FUNCTION_BLOCK FB_TIIAlarm
VAR_INPUT
	vIO							: ST_TCMultiLevel_VIO;
	stTCColVIO					: ST_TCColumn_VIO;
	NoOfTIIAlm					: INT	:= NO_OF_TII_SENSOR;
	iLevel						: INT	:= 1;
END_VAR

VAR_OUTPUT
	isTIIError					: BOOL;
	TIIAlarmLED					: BOOL;
	TIIAlarmEPT					: BOOL;
	iUnBlock					: DINT;
	isAboveCellLeakage			: BOOL;
END_VAR

VAR
	DIFU						: R_TRIG;
	tim							: TON;
	delay						: FB_Delay;
	tPOn						: BOOL;	//testerPowerOutoutOn after Delay
	dPOn						: BOOL; //dpsPwrbit after Delay
	bitNo						: INT;
	almRset						: BOOL;
	
	ArrAlmBitBefDelay			: ARRAY[1..NO_OF_TII_SENSOR] OF BOOL;
	ArrAlmBitAftDelay			: ARRAY[1..NO_OF_TII_SENSOR] OF BOOL;
	ArrAlarmKeepBit				: ARRAY[1..NO_OF_TII_SENSOR] OF BOOL;
	ArrDelayAlarm				: ARRAY[1..NO_OF_TII_SENSOR] OF FB_AlarmDelay;
	Arr_ms						: ARRAY[1..NO_OF_TII_SENSOR] OF INT;
	bTIIByPassArray				: ARRAY[1..NO_OF_TII_SENSOR] OF BOOL;
	i							: INT;
	bTest						: BOOL;
	delayExtTimeOut				: FB_Delay;
	delayRetTimeOut				: FB_Delay;
	delayDrawerUpTimeOut		: FB_Delay;
	delayDrawerDownTimeOut		: FB_Delay;
	//iUnBlock:INT;
	alarmReset					: BOOL;  //1: reset timer when alarm reset, 0: do not reset timer
END_VAR

VAR_IN_OUT
	
	//bLibError : BOOL;
	//stAlmSubMod:ST_AlarmSubmodules;
	//stAlmMod:ST_AlarmModules;
END_VAR

//<HMI_TII_Test>

IF bHMITIIBypass THEN
	bTIIByPassArray							:= stHMITIIByPassArray[iLevel].bHMITIIByPassArray;
	//FOR i:=1 TO NoOfTIIAlm DO
	//	bTIIByPassArray[i]:= NOT stHMITIIByPassArray[iLevel].bHMITIIByPassArray[i];
	//END_FOR
ELSE
	FOR i := 1 TO NoOfTIIAlm DO
		//bTIIByPassArray[i]:=bEnableTIIAlarm;
		 bTIIByPassArray[i]					:= TC_ModuleState[iLevel].TCSite[1].TIERII = E_State.eEnabled;
	END_FOR
END_IF
//</HMI_TII_Test>
//IF bTest THEN
AlarmUpdate(bENs:= bTIIByPassArray);
//END_IF

METHOD AlarmUpdate : BOOL
VAR_INPUT
	bENs 					: ARRAY [1..NO_OF_TII_SENSOR] OF BOOL;
END_VAR

VAR_OUTPUT
END_VAR

VAR_IN_OUT
	//ArrAlarmKeepBit:ST_AlarmTags;
END_VAR

VAR
	_bError					: BOOL;
	bTstOnCmd 				: BOOL;
	bChkTstOn 				: BOOL;
	bAPOnCmd				: BOOL;
	bChkAPOn 				: BOOL;
	drawerExtendOutput		: BOOL; // Condition
	drawerRetractOutput		: BOOL; // Condition
	drawerUpOutput			: BOOL;
	drawerDownOutput		: BOOL;
	
	i						: INT;
	j						: INT;
	iSysAlarmID 			: INT;
	e						: E_TIIAlarm;
END_VAR
IF iLevel = 0 THEN
	RETURN;
END_IF

//FB_M_nCyclic_tSensorTimeOut
DIFU(
	CLK 																:= vIO.ipTesterPowerOn);
	                                                					
tim(                                                					
	IN 																	:= TRUE,
	PT																	:= INT_TO_TIME(1000));
	                                                					
tPOn 																	:=	VIO.bTstDelInt; //Delay and TesterPwrOnOutput
                                                    					
delay(                                              					
	msec 																:= 100,
	in 																	:= tPOn, 
	out 																:= dPOn);
	                                                					
delayExtTimeOut(                                    	
	msec																:= TIME_TO_INT(tDwrCylExtRetTimeOut),
	in																	:= vIO.opCellDrawerCylExtend,
	out																	:= drawerExtendOutput);
	                                                					
delayRetTimeOut(                                    					
	msec																:= TIME_TO_INT(tDwrCylExtRetTimeOut),
	in																	:= vIO.opCellDrawerCylRetract,
	out																	:= drawerRetractOutput);
	

delayDrawerUpTimeOut(
	msec																:= TIME_TO_INT(tDwrCylUpDownTimeOut),
	in																	:= vIO.opCellDrawerCylUp,
	out																	:= drawerUpOutput);

delayDrawerDownTimeOut(
	msec																:= TIME_TO_INT(tDwrCylUpDownTimeOut),
	in																	:= vIO.opCellDrawerCylDown,
	out																	:= drawerDownOutput);
	

//lRt:= FALSE; //:=AP_Deactuated(if AP Down Can Retract)
//lEt:= FALSE;
bTstOnCmd																:= vIO.bDPSPowerOnOff;
bChkTstOn																:= vIO.bChkTesterOn;
bAPOnCmd																:= vIO.bAP240ACPowerOnOff;
bChkAPOn																:= vIO.bChkAP240On;


//Auto reset Door lock alarm
IF ALMTC.Level[iLevel].AlarmID[E_TIIAlarm.ipTCCellDoorClosed] AND vIO.ipTCCellDoorClosed THEN
	ALMTC.Level[iLevel].AlarmID[E_TIIAlarm.ipTCCellDoorClosed]			:= FALSE;
END_IF

IF ALMTC.Level[iLevel].AlarmID[E_AlarmID.DoorCloseSignalNotDetected] AND vIO.ipTCCellDoorOpenCloseStatus THEN
	ALMTC.Level[iLevel].AlarmID[E_AlarmID.DoorCloseSignalNotDetected]			:= FALSE;
END_IF

//Auto reset Door lock alarm (Debugcart only)
IF bDebugCart THEN
	//auto clear alarm if door is closed 
	IF ALMTC.Level[iLevel].AlarmID[E_AlarmID.TBotSideDoorCloseSignalNotDetected] THEN
		IF VIO.ipTCCellTbotSideDoorOpenCloseStatus01 AND VIO.ipTCCellTbotSideDoorOpenCloseStatus02 THEN
			ALMTC.Level[iLevel].AlarmID[E_AlarmID.TBotSideDoorCloseSignalNotDetected]		:= FALSE;
		END_IF
	END_IF
	
	//auto clear alarm if door is locked
	IF ALMTC.Level[iLevel].AlarmID[E_TIIAlarm.FrontDoorLockSignalNotDetected] THEN
		IF VIO.ipTCCellTbotSideDoorLocked01 AND VIO.ipTCCellTbotSideDoorLocked02 THEN
			ALMTC.Level[iLevel].AlarmID[E_TIIAlarm.FrontDoorLockSignalNotDetected]		:= FALSE;
		END_IF
	END_IF
END_IF


FOR i := 1 TO NoOfTIIAlm DO	
	CASE i OF
		(*E_TIIAlarm.ipAPPresentSensor: 
			e															:= E_TIIAlarm.ipAPPresentSensor; 
			ArrAlmBitBefDelay[E_TIIAlarm.ipAPPresentSensor]				:= (NOT	vIO.ipAPPresentSensor) AND bENs[1];  		
			Arr_ms[e] 													:= 500;  (*TIIAlmText[e]:='AP_PresentSensor'*); //****stTCVIO.iAlarmCode=  E_Alarm.ipAP_PresentSensor 	 ;*)
			
        E_TIIAlarm.ipAPPowerOn: 
			e															:= E_TIIAlarm.ipAPPowerOn; 
			ArrAlmBitBefDelay[E_TIIAlarm.ipAPPowerOn]					:= (NOT vIO.ipAPPowerOn) AND VIO.ipAPPresentSensor AND GVL_DUT_TC_AP240ACPower.Failed AND bENs[2];
			Arr_ms[e] 													:= 500;  (*TIIAlmText[e]:='AP_PowerOn'*); 
			
	    E_TIIAlarm.ipAPReady: 
			e															:= E_TIIAlarm.ipAPReady; 
			ArrAlmBitBefDelay[E_TIIAlarm.ipAPReady]						:= (NOT vIO.ipAPReady) AND vIO.ipAPPresentSensor AND bENs[3]; 	
			Arr_ms[e] 													:= 500;  (*TIIAlmText[e]:='AP_Ready' 		    	*);      
			
	    (*E_TIIAlarm.ipAPDeactuatedPLC: 
			e															:= E_TIIAlarm.ipAPDeactuatedPLC; 
			ArrAlmBitBefDelay[E_TIIAlarm.ipAPDeactuatedPLC]				:= (NOT vIO.ipHandlerSafeToEnterPLC) AND vIO.ipAPPresentSensor AND bENs[4]; 			
			Arr_ms[e] 													:= 500;  (*TIIAlmText[e]:='AP_DeactuatedPLC'*); *)
  
	    (*E_TIIAlarm.ipAPDeactuatedHwr: 
			e															:= E_TIIAlarm.ipAPDeactuatedHwr; 
			ArrAlmBitBefDelay[E_TIIAlarm.ipAPDeactuatedHwr]				:= (NOT	vIO.ipHandlerSafeToEnterHwr) AND vIO.ipAPPresentSensor AND bENs[5]; 			
			Arr_ms[e] 													:= 500;  (*TIIAlmText[e]:='AP_DeactuatedHwr'*); *)
			
	    E_TIIAlarm.ipCellFluidLeakage1: 
			e															:= E_TIIAlarm.ipCellFluidLeakage1; 
			ArrAlmBitBefDelay[E_TIIAlarm.ipCellFluidLeakage1]			:= vIO.ipCellFluidLeakage1 (*AND bENs[6]*); 			
			Arr_ms[e] 													:= 500;  (*TIIAlmText[e]:='CellFluidLeakage1' 	*);   
			
	    E_TIIAlarm.ipCellFluidLeakage2: 
			e															:= E_TIIAlarm.ipCellFluidLeakage2; 
			ArrAlmBitBefDelay[E_TIIAlarm.ipCellFluidLeakage2]			:= vIO.ipCellFluidLeakage2 (*AND bENs[7]*) ; 			
			Arr_ms[e] 													:= 500;  (*TIIAlmText[e]:='CellFluidLeakage2'*);   
			
	    E_TIIAlarm.ipCellGroundFault: 
			e															:= E_TIIAlarm.ipCellGroundFault; 
			ArrAlmBitBefDelay[E_TIIAlarm.ipCellGroundFault]				:= vIO.ipCellGroundFault AND bENs[8]; 			
			Arr_ms[e] 													:= 500;  (*TIIAlmText[e]:='CellGroundFault'*);
			
        (*E_TIIAlarm.ipTesterPresent: 
			e															:= E_TIIAlarm.ipTesterPresent; 
			ArrAlmBitBefDelay[E_TIIAlarm.ipTesterPresent]				:= (NOT	vIO.ipTesterPresent) AND bENs[9]; 			
			Arr_ms[e] 													:= 500;  (*TIIAlmText[e]:='TesterPresent'*);*)
			
        E_TIIAlarm.ipTesterPowerOn: 
			e															:= E_TIIAlarm.ipTesterPowerOn; 
			ArrAlmBitBefDelay[E_TIIAlarm.ipTesterPowerOn]				:= (NOT	vIO.ipTesterPowerOn) AND vIO.ipTesterPresent AND bChkTstOn AND bENs[10]; 			
			Arr_ms[e] 													:= 500;  (*TIIAlmText[e]:='TesterPowerOn'*);
    
        (*E_TIIAlarm.ipTesterReady: 
			e															:= E_TIIAlarm.ipTesterReady; 
			ArrAlmBitBefDelay[E_TIIAlarm.ipTesterReady]					:= (NOT	vIO.ipTesterReady) AND vIO.ipTesterPresent AND bENs[11]; 	
			Arr_ms[e] 													:= 500;  (*TIIAlmText[e]:='TesterReady'*);*)
			   
       	E_TIIAlarm.ipTCCellDoorClosed: 
			stTCColVIO													:= fbTCColumn.P_stTCColumnVIO;
			e															:= E_TIIAlarm.ipTCCellDoorClosed; 
			ArrAlmBitBefDelay[E_TIIAlarm.ipTCCellDoorClosed]			:= (NOT	vIO.ipTCCellDoorClosed) AND stTCColVIO.ipTbotDoorClosedSignal; //AND bENs[12]; 							
			Arr_ms[e] 													:= 500;  (*TIIAlmText[e]:='TCCellDoorClosed' *);
			
        E_TIIAlarm.ipTesterLatchesClosed: 
			e															:= E_TIIAlarm.ipTesterLatchesClosed ; 
			ArrAlmBitBefDelay[E_TIIAlarm.ipTesterLatchesClosed]			:= (NOT	vIO.ipTesterLatchesClosed) AND (bTstOnCmd OR vIO.ipTesterPresent) AND bENs[13] ; 
			Arr_ms[e] 													:= 500;  (*TIIAlmText[e]:='TesterLatchesClosed'*);
			
        (*E_TIIAlarm.ipTIUPresent: 
			e															:= E_TIIAlarm.ipTIUPresent; 
			ArrAlmBitBefDelay[E_TIIAlarm.ipTIUPresent]					:= (NOT	vIO.ipTIUPresent) AND bENs[14]; 						
			Arr_ms[e] 													:= 500;  (*TIIAlmText[e]:='TIUPresent'*);*)
			
        E_TIIAlarm.TBOT_TC_ACPower_Signal: 
			e															:= E_TIIAlarm.TBOT_TC_ACPower_Signal; 
			ArrAlmBitBefDelay[E_TIIAlarm.TBOT_TC_ACPower_Signal]		:= (vIO.TBOT_TC_ACPower_Signal) AND (NOT bDebugCart) AND (NOT bDebugStation) AND bENs[14]; 
			Arr_ms[e] 													:= 500;  (*TIIAlmText[e]:='TCDrawerCylRetractRS'*);
			
		E_TIIAlarm.DS_Facility_EAP_ACPower_Signal: 
			e																:= E_TIIAlarm.DS_Facility_EAP_ACPower_Signal; 
			ArrAlmBitBefDelay[E_TIIAlarm.DS_Facility_EAP_ACPower_Signal]	:= bDebugCart AND DS_Facility_eapShutOffAllACPower AND bENs[15]; 							
			Arr_ms[e] 														:= 500;  (*TIIAlmText[e]:='DS_Facility_EAP_ACPower_Signal' *);
			
      	E_TIIAlarm.FrontDoorLockSignalNotDetected: 
			e																:= E_TIIAlarm.FrontDoorLockSignalNotDetected; 
			ArrAlmBitBefDelay[E_TIIAlarm.FrontDoorLockSignalNotDetected]	:= bDebugCart AND ((NOT vIO.ipTCCellTbotSideDoorLocked01) OR (NOT vIO.ipTCCellTbotSideDoorLocked02)); //AND bENs[16]; 							
			Arr_ms[e] 														:= 500;  (*TIIAlmText[e]:='ipTCCellTbotSideDoorLocked01' *);	
					
        E_TIIAlarm.ipTCDrawerExtendSignal: 
			e																:= E_TIIAlarm.ipTCDrawerExtendSignal; 
			ArrAlmBitBefDelay[E_TIIAlarm.ipTCDrawerExtendSignal]			:= (NOT	vIO.ipTCDrawerCylExtendRS) AND (*vIO.opTesterDrawerAirSupplySol AND	vIO.opCellDrawerCylExtend AND*) (NOT bDebugCart) AND drawerExtendOutput AND bENs[15]; 
			Arr_ms[e] 														:= 500;  (*TIIAlmText[e]:='TCDrawerCylExtendRS'*);
			
        E_TIIAlarm.ipTCDrawerRetractSignal: 
			e																:= E_TIIAlarm.ipTCDrawerRetractSignal; 
			ArrAlmBitBefDelay[E_TIIAlarm.ipTCDrawerRetractSignal]			:= (NOT	vIO.ipTCDrawerCylRetractRS) AND (*vIO.opTesterDrawerAirSupplySol AND vIO.opCellDrawerCylRetract AND*) drawerRetractOutput AND bENs[16]; 
			Arr_ms[e] 														:= 500;  (*TIIAlmText[e]:='TCDrawerCylRetractRS'*);	
		
		E_TIIAlarm.ipTCDrawerUpSignal:
			e																:= E_TIIAlarm.ipTCDrawerUpSignal;
			ArrAlmBitBefDelay[E_TIIAlarm.ipTCDrawerUpSignal]				:= (NOT	vIO.ipTCDrawerCylUpRS) AND drawerUpOutput AND bENs[16]; 
			Arr_ms[e] 														:= 500;  (*TIIAlmText[e]:='TCDrawerCylupRS'*);	
		
		E_TIIAlarm.ipTCDrawerDownSignal:
			e																:= E_TIIAlarm.ipTCDrawerUpSignal;
			ArrAlmBitBefDelay[E_TIIAlarm.ipTCDrawerDownSignal]				:= (NOT	vIO.ipTCDrawerCylDownRS) AND drawerDownOutput AND bENs[16]; 
			Arr_ms[e] 														:= 500;  (*TIIAlmText[e]:='TCDrawerCyldownRS'*);
			
	END_CASE

	//Delay Library for all alarm bits
	ArrDelayAlarm[i](
		alarmState															:= ArrAlmBitBefDelay[i],
		alarmResetTimer														:= alarmReset,
		triggerAlarmState													=> ArrAlmBitAftDelay[i],
		msec																:= Arr_ms[i]);

	 //Trigger alarm if alarm state delay time expired.
	IF ArrAlmBitAftDelay[i] THEN
		ALMTC.Level[iLevel].AlarmID[i]									:= TRUE;
	END_IF
		
	isTIIError															:= ALMTC.Level[iLevel].AlarmID[i];
END_FOR

alarmReset			:= FALSE;	//false back and wait for next alarm reset to reset alarm timer.


//////////////////////////////////////////////////////////////////////////////////////////////////////////////////////////////////////////////////////////////////////////////////////////////////////////////////////////////////////////////////////
//////////////////////// TIIAlarmLED : Trigger EPT state alarms ////////////////////////
//////////////////////// TIIAlarmEPT : Trigger AlarmLED alarms	////////////////////////
//////////////////////////////////////////////////////////////////////////////////////////////////////////////////////////////////////////////////////////////////////////////////////////////////////////////////////////////////////////////////////

//Check Above cell whether has leakage alarm
isAboveCellLeakage		:= M_AboveLeakageChecking(currentLevel	:= iLevel);
																			
TIIAlarmLED																:=	ALMTC.Level[iLevel].AlarmID[E_TIIAlarm.ipAPPowerOn 		   	   			]   OR 
		    																ALMTC.Level[iLevel].AlarmID[E_TIIAlarm.ipAPReady		       	   		]   OR
																			ALMTC.Level[iLevel].AlarmID[E_TIIAlarm.ipTesterLatchesClosed    		]	OR
																			ALMTC.Level[iLevel].AlarmID[E_TIIAlarm.ipTesterPowerOn	       			]   OR
																			ALMTC.Level[iLevel].AlarmID[E_TIIAlarm.ipTesterReady	           		]   OR
																			ALMTC.Level[iLevel].AlarmID[E_TIIAlarm.ipTCCellDoorClosed	   			]   OR
																			ALMTC.Common.AlarmID[E_ColAlarm.ipTbotDoorClosedSignal					]	OR
																			ALMTC.Level[iLevel].AlarmID[E_TIIAlarm.ipCellFluidLeakage1	   			]   OR
																			ALMTC.Level[iLevel].AlarmID[E_TIIAlarm.ipCellFluidLeakage2	   			]   OR
																			ALMTC.Level[iLevel].AlarmID[E_TIIAlarm.ipCellGroundFault 	   			]   OR
																			ALMTC.Level[iLevel].ALarmID[E_AlarmID.DrawerDownError					]	OR
																			ALMTC.Level[iLevel].ALarmID[E_AlarmID.DrawerUpError						]	OR
																			ALMTC.Level[iLevel].ALarmID[E_AlarmID.DrawerExtendError					]	OR
																			ALMTC.Level[iLevel].ALarmID[E_AlarmID.DrawerRetractError				]	OR
																			ALMTC.Level[iLevel].ALarmID[E_AlarmID.APIsNotInUPPosition				]	OR
																			ALMTC.Common.AlarmID[E_ColAlarm.ipColumnFluid_PCW_Leakage				]	OR
																			ALMTC.Level[iLevel].AlarmID[E_TIIAlarm.FrontDoorLockSignalNotDetected	]	OR
																			ALMTC.Level[iLevel].AlarmID[E_TIIAlarm.TBOT_TC_ACPower_Signal   		] 	OR	
																			ALMTC.Level[iLevel].AlarmID[E_TIIAlarm.DS_Facility_EAP_ACPower_Signal	]	OR
																			ALMTC.Level[iLevel].AlarmID[E_TIIAlarm.ipTCDrawerExtendSignal			]	OR
																			ALMTC.Level[iLevel].AlarmID[E_TIIAlarm.ipTCDrawerRetractSignal			]	OR
																			ALMTC.Level[iLevel].AlarmID[E_TIIAlarm.ipTCDrawerUpSignal				]	OR
																			ALMTC.Level[iLevel].AlarmID[E_TIIAlarm.ipTCDrawerDownSignal				]	OR
																			isAboveCellLeakage;
																			
																			
TIIAlarmEPT																:= 	ALMTC.Level[iLevel].AlarmID[E_TIIAlarm.ipAPPowerOn						]	OR
																			ALMTC.Level[iLevel].AlarmID[E_TIIAlarm.ipAPReady						]	OR
																			ALMTC.Level[iLevel].AlarmID[E_TIIAlarm.ipTesterLatchesClosed			]	OR
																			ALMTC.Level[iLevel].AlarmID[E_AlarmID.DrawerRetractError				]	OR
																			ALMTC.Level[iLevel].AlarmID[E_AlarmID.DrawerExtendError					]	OR
																			ALMTC.Level[iLevel].AlarmID[E_TIIAlarm.ipTCCellDoorClosed				]	OR
																			ALMTC.Level[iLevel].AlarmID[E_TIIAlarm.ipCellGroundFault				]	OR
																			ALMTC.Level[iLevel].AlarmID[E_TIIAlarm.ipCellFluidLeakage1				]	OR
																			ALMTC.Level[iLevel].AlarmID[E_TIIAlarm.ipCellFluidLeakage2				]	OR
																			ALMTC.Common.AlarmID[E_ColAlarm.ipColumnFluid_PCW_Leakage				]	OR
																			ALMTC.Common.AlarmID[E_ColAlarm.ipTbotDoorClosedSignal					]	OR
																			ALMTC.Level[iLevel].AlarmID[E_TIIAlarm.FrontDoorLockSignalNotDetected	]	OR
																			ALMTC.Level[iLevel].AlarmID[E_TIIAlarm.TBOT_TC_ACPower_Signal   		]	OR
																			ALMTC.Level[iLevel].AlarmID[E_TIIAlarm.DS_Facility_EAP_ACPower_Signal	]	OR
																			ALMTC.Level[iLevel].AlarmID[E_TIIAlarm.ipTCDrawerExtendSignal			]	OR
																			ALMTC.Level[iLevel].AlarmID[E_TIIAlarm.ipTCDrawerRetractSignal			]	OR
																			ALMTC.Level[iLevel].AlarmID[E_TIIAlarm.ipTCDrawerUpSignal				]	OR
																			ALMTC.Level[iLevel].AlarmID[E_TIIAlarm.ipTCDrawerDownSignal				]	OR
																			isAboveCellLeakage;
END_METHOD

METHOD M_AboveLeakageChecking : BOOL
VAR_INPUT
	currentLevel	: INT;
END_VAR
VAR
	maxLevel		: INT;
END_VAR
maxLevel									:= NO_OF_LEVEL;

IF currentLevel = maxLevel THEN
	M_AboveLeakageChecking						:= FALSE;
	RETURN;
END_IF

IF ALMTC.Level[currentLevel+1].AlarmID[E_TIIAlarm.ipCellFluidLeakage1] OR ALMTC.Level[currentLevel+1].AlarmID[E_TIIAlarm.ipCellFluidLeakage2] THEN
	M_AboveLeakageChecking					:= TRUE;
ELSIF ALMTC.Level[currentLevel+2].AlarmID[E_TIIAlarm.ipCellFluidLeakage1] OR ALMTC.Level[currentLevel+2].AlarmID[E_TIIAlarm.ipCellFluidLeakage2] THEN
	M_AboveLeakageChecking					:= TRUE;
END_IF
END_METHOD

PROPERTY P_ErrClear : BOOL
GET
END_GET
SET
alarmReset	:= P_ErrClear;
END_SET
END_PROPERTY

END_FUNCTION_BLOCK

(* stored: Version 1.1.0.1, ProductVersion 3.1.4022.18
   POU FB_TIIAlarm: Id {0b288081-bd94-440a-8fe6-c5b6955eac6e}, SpecialFunc None
   Method AlarmUpdate: Id {397002b7-185c-4e8e-b452-1b3a6b84eaa4}
   Method M_AboveLeakageChecking: Id {0b729bd7-55a1-4289-91e6-7b49f3713973}
   Property P_ErrClear: Id {a7ea7319-566b-4b4c-a0be-fa28aa059c11}
   Get Get: Id {423550e5-8c77-479e-a2f2-c9a4c635ec9f}
   Set Set: Id {a6fac879-a371-480d-9d97-36ad329adf11} *)
